// TwinCAT 3 PLC project PLC1
// Title: TcHAL
// Company: none
// Author: Tobias Freyermuth
// ProjectVersion: 0.1.4
// Description: Hardware Abstraction Layer of TwinCAT fieldbus devices
// ProgramVersion: 3.1.4024.12
// libraries:
//   Tc2_EtherCAT, * (Beckhoff Automation GmbH)
//   Tc2_Standard, * (Beckhoff Automation GmbH)
//   Tc2_System, * (Beckhoff Automation GmbH)
//   Tc2_Utilities, * (Beckhoff Automation GmbH)
//   Tc3_Module, * (Beckhoff Automation GmbH)
//   TcUnit, * (www.tcunit.org)
// project tree:
//   analog_input/temperature/ EL3202_0010.TcPOU
//   analog_input/voltage/ EL3164.TcPOU
//   analog_input/_internal/ AI_Channel.TcPOU, AI_Voltage_Channel.TcPOU, AI_Temperature_Channel.TcPOU, I_AI_percentage.TcIO (not stored), I_AI_Temperature.TcIO (not stored), I_AI_Voltage.TcIO (not stored)
//   analog_output/voltage/ EL4002.TcPOU (not stored), EL4102.TcPOU (not stored), EL4004.TcPOU (not stored), EL4134.TcPOU (not stored)
//   analog_output/_internal/ AO_Voltage_Channel.TcPOU (not stored), I_AO_Voltage.TcIO (not stored)
//   coupler/ EK1101.TcPOU (not stored)
//   digital_input/ EL1008.TcPOU (not stored), EL1104.TcPOU (not stored), EL1144.TcPOU (not stored), EL1808.TcPOU (not stored), EL1124.TcPOU (not stored), EL1809.TcPOU (not stored)
//   digital_input/_internal/ HAL_DI_Channel.TcPOU (not stored), I_HAL_DI.TcIO (not stored)
//   digital_output/ EL2008.TcPOU (not stored), EL2124.TcPOU (not stored), EL2024_0010.TcPOU (not stored), EL2502.TcPOU (not stored) (excluded from build), EL2595.TcPOU (not stored), EL2612.TcPOU (not stored), EL2521.TcPOU (not stored) (excluded from build), EL2004.TcPOU (not stored), EL2634.TcPOU (not stored), EL2808.TcPOU (not stored), EL2624.TcPOU (not stored), EL2794.TcPOU (not stored)
//   digital_output/_internal/ HAL_DO_Channel.TcPOU (not stored), I_HAL_DO.TcIO (not stored)
//   / HAL_ErrorEnum.TcDUT (not stored), MAIN.TcPOU (not stored), PlcTask.TcTTO (not stored), Settings.TcGVL (not stored), _internal.TcGVL (not stored)
//   InterfaceManager/ InterfaceManager.TcPOU (not stored), InterfaceManager_test.TcPOU (not stored), I_AI_Percentage_register.TcDUT (not stored), I_AO_Voltage_register.TcDUT (not stored), I_AI_Voltage_register.TcDUT (not stored), I_InterfaceManager.TcIO (not stored)
//   Project Information/ F_GetCompany.TcPOU (not stored), F_GetTitle.TcPOU (not stored), F_GetVersion.TcPOU (not stored)
//   Version/ Global_Version.TcGVL (not stored)
//   _internal/CoE/BeckhoffTerminalConfigEnums/ ENU_DT0800EN02.TcDUT (not stored), ENU_DT0801EN03.TcDUT (not stored)
//   _internal/CoE/buffer/ ring_buffer_CoE_read.TcPOU (not stored)
//   _internal/CoE/ CoE_communication_handler.TcPOU, CoE_property_handler.TcPOU (not stored), CoE_UML_Class Diagram.TcCD (not stored), I_CoE_config_common.TcIO (not stored), I_CoE_property.TcIO, I_CoE_communication_handler.TcIO (not stored)
//   _internal/CoE/properties/ CoE_property.TcPOU
//   _internal/ I_device_control.TcIO (not stored), I_terminal_execution.TcIO (not stored), I_coupler_execution.TcIO (not stored), linear_adc_to_phy.TcPOU (not stored), linear_phy_to_adc.TcPOU (not stored), linear_phy_to_adc_test.TcPOU (not stored), linear_adc_to_phy_test.TcPOU (not stored)

// ---- _internal/CoE/I_CoE_property.TcIO
INTERFACE I_CoE_property

PROPERTY CoE_communication_handler : I_CoE_communication_handler
GET
END_GET
SET
END_SET
END_PROPERTY

PROPERTY dataTypeSize : UDINT
GET
END_GET
END_PROPERTY

METHOD get_value : BOOL
VAR_OUTPUT
    value : Tc2_Utilities.T_Arg ;
	errId : UDINT;
END_VAR
END_METHOD

METHOD handle_read_callback : BOOL
VAR_INPUT
	pt_buffer : POINTER TO Tc2_Utilities.T_Arg;
	errId : UDINT;
END_VAR
END_METHOD

METHOD handle_write_callback : BOOL
VAR_INPUT
	errId : UDINT;
END_VAR
END_METHOD

PROPERTY Index : word
GET
END_GET
END_PROPERTY

PROPERTY init_done : bool
GET
END_GET
END_PROPERTY

PROPERTY PropertyType : E_ArgType
GET
END_GET
SET
END_SET
END_PROPERTY

(**
This method is initializing or reinitializing the property and returns TRUE when this is done.
In case of an error during the init it returns the ErrorCode related to the error that occurred.
*)
METHOD reinit : BOOL
VAR_OUTPUT
	errId: UDINT;
END_VAR
END_METHOD

METHOD run : BOOL
VAR_INPUT
END_VAR
END_METHOD

METHOD set_value : BOOL
VAR_INPUT
    value : Tc2_Utilities.T_Arg ;
END_VAR
END_METHOD

PROPERTY SlaveAddress : UINT
GET
END_GET
SET
END_SET
END_PROPERTY

PROPERTY SubIndex : BYTE
GET
END_GET
END_PROPERTY

PROPERTY valueToWrite : Tc2_Utilities.T_Arg
GET
END_GET
END_PROPERTY

END_INTERFACE

// ---- analog_input/temperature/EL3202_0010.TcPOU
FUNCTION_BLOCK EL3202_0010 IMPLEMENTS I_terminal_execution
VAR_INPUT
END_VAR
VAR_OUTPUT
	AI_Temperature_channel_1 		: I_AI_Temperature :=_channel_1;
	AI_Temperature_channel_2 		: I_AI_Temperature :=_channel_2;
	AI_percent_channe_1				: I_AI_percentage := _channel_1;
	AI_percent_channe_2				: I_AI_percentage := _channel_2;
END_VAR
VAR
// == IO Mapping ==============================================================
	WcState_WcState			AT%I*: BOOL;
	InfoData_State			AT%I*: UINT;
	InfoData_AdsAddr_netId  AT%I*: AMSNETID;
	InfoData_AdsAddr_port 	AT%I*: WORD;
	
	// Channel 1
	RTD_Inputs_Channel_1_Value        			AT%I*: INT;	
	RTD_Inputs_Channel_1_Status_Underrange   	AT%I*: BOOL;
	RTD_Inputs_Channel_1_Status_Overrange   	AT%I*: BOOL;
	RTD_Inputs_Channel_1_Status_Limit_1   		AT%I*: BYTE;
	RTD_Inputs_Channel_1_Status_Limit_2   		AT%I*: BYTE;
	RTD_Inputs_Channel_1_Status_Error   		AT%I*: BOOL;
	RTD_Inputs_Channel_1_Status_TxPDO_State   	AT%I*: BOOL;
	RTD_Inputs_Channel_1_Status_TxPDO_Toggle   	AT%I*: BOOL;
	
	// Channel 2
	RTD_Inputs_Channel_2_Value        			AT%I*: INT;	
	RTD_Inputs_Channel_2_Status_Underrange   	AT%I*: BOOL;
	RTD_Inputs_Channel_2_Status_Overrange   	AT%I*: BOOL;
	RTD_Inputs_Channel_2_Status_Limit_1   		AT%I*: BYTE;
	RTD_Inputs_Channel_2_Status_Limit_2   		AT%I*: BYTE;
	RTD_Inputs_Channel_2_Status_Error   		AT%I*: BOOL;
	RTD_Inputs_Channel_2_Status_TxPDO_State   	AT%I*: BOOL;
	RTD_Inputs_Channel_2_Status_TxPDO_Toggle   	AT%I*: BOOL;
// ============================================================================

	_channel_1 : AI_Temperature_Channel(adc_min:=ADC_MIN, adc_max:=ADC_MAX, physical_min:=PHYSICAL_MIN, physical_max:=PHYSICAL_MAX, channel_number:=1);
	_channel_2 : AI_Temperature_Channel(adc_min:=ADC_MIN, adc_max:=ADC_MAX, physical_min:=PHYSICAL_MIN, physical_max:=PHYSICAL_MAX, channel_number:=2);

    
	// ===============================================================================
	// CoE handling  
	// ==============
    _I_CoE_com_handler      : I_CoE_communication_handler;
    _CoE_prop_handler       : CoE_property_handler;
    // ====  CoE properties  ===========
	_p_DeviceName 			: CoE_property(Index:=16#1008 , SubIndex:=0,PropertyType:=Tc2_Utilities.ARGTYPE_STRING, writable:=FALSE, propertyPullMode:=0, pollingInterval:=T#5S);
	_p_DeviceType 			: CoE_property(Index:=16#1000 , SubIndex:=0,PropertyType:=Tc2_Utilities.ARGTYPE_UDINT, writable:=FALSE, propertyPullMode:=0, pollingInterval:=T#5S);
	_p_ProductCode 			: CoE_property(Index:=16#1018 , SubIndex:=2,PropertyType:=Tc2_Utilities.ARGTYPE_UDINT, writable:=FALSE, propertyPullMode:=0, pollingInterval:=T#5S);
	_p_Revision 			: CoE_property(Index:=16#1018 , SubIndex:=3,PropertyType:=Tc2_Utilities.ARGTYPE_UDINT, writable:=FALSE, propertyPullMode:=0, pollingInterval:=T#5S);
	_p_SerialNumber 		: CoE_property(Index:=16#1018 , SubIndex:=4,PropertyType:=Tc2_Utilities.ARGTYPE_UDINT, writable:=FALSE, propertyPullMode:=0, pollingInterval:=T#5S);
	_p_SoftwareVersion		: CoE_property(Index:=16#100A , SubIndex:=0,PropertyType:=Tc2_Utilities.ARGTYPE_STRING, writable:=FALSE, propertyPullMode:=0, pollingInterval:=T#5S);
	_p_VendorId 			: CoE_property(Index:=16#1018 , SubIndex:=1,PropertyType:=Tc2_Utilities.ARGTYPE_UDINT, writable:=FALSE, propertyPullMode:=0, pollingInterval:=T#5S);
	_p_HardwareVersion		: CoE_property(Index:=16#1009 , SubIndex:=0,PropertyType:=Tc2_Utilities.ARGTYPE_STRING, writable:=FALSE, propertyPullMode:=0, pollingInterval:=T#5S);
	// ==============
	_properties  : ARRAY[1..8]OF I_CoE_property:=[
		_p_DeviceName, _p_DeviceType, _p_ProductCode, _p_Revision, _p_SerialNumber, 
		_p_SoftwareVersion, _p_VendorId, _p_HardwareVersion
	];
	// ===============================================================================
    
    
	_I_InterfaceManager : I_InterfaceManager;
	_terminal_name      : STRING;
	reg_errId           : HAL_ErrorEnum;
	_InitState          : INT;
    neg_wcState: f_trig;
END_VAR
VAR CONSTANT
	ADC_MIN        	: INT:=0;
	ADC_MAX        	: INT:=32767;
	PHYSICAL_MIN 	: INT:=0;
	PHYSICAL_MAX 	: INT:=10;
	
    HARDWARE_REVSION : UINT:=19;
END_VAR

CASE _InitState OF 
	0:  // init parent
        IF _I_InterfaceManager <> 0 AND 
            _I_CoE_com_handler <> 0
        THEN
            _InitState := 5;
		END_IF
		
	5: 
		IF NOT _I_InterfaceManager.register_terminal(terminal_name:=_terminal_name , errId=>reg_errId ) THEN
			RETURN;
		ELSE
			_InitState := 10;
		END_IF
        
	10: // register channel 1 percentage interface 
		IF _I_InterfaceManager.register_I_AI_Percentage(_channel_1, _terminal_name, channel_number := 1, errId=>reg_errId) THEN 
			_InitState := 20;
		END_IF
	20: // register channel 2 percentage interface 
		IF _I_InterfaceManager.register_I_AI_Percentage(_channel_2, _terminal_name, channel_number := 2, errId=>reg_errId) THEN 
			_InitState := 30;
		END_IF

	30: // register channel 1 voltage interface 
		IF _I_InterfaceManager.register_I_AI_Percentage(_channel_1, _terminal_name, channel_number := 1, errId=>reg_errId) THEN 
			_InitState := 40;
		END_IF
		
	40: // register channel 2 voltage interface 
		IF _I_InterfaceManager.register_I_AI_Percentage(_channel_2, _terminal_name, channel_number := 2, errId=>reg_errId) THEN 
			_InitState := 50;
		END_IF
ELSE
	// Channel 1
	_channel_1.wcState							:= WcState_WcState;
	_channel_1.terminal_value 					:= RTD_Inputs_Channel_1_Value;
	_channel_1.io_status_Underrange 			:= RTD_Inputs_Channel_1_Status_Underrange;
	_channel_1.io_status_Overrange 				:= RTD_Inputs_Channel_1_Status_Overrange;
	_channel_1.io_status_Limit_1_greater_value 	:= RTD_Inputs_Channel_1_Status_Limit_1.0;
	_channel_1.io_status_Limit_1_smaller_value	:= RTD_Inputs_Channel_1_Status_Limit_1.1;
	_channel_1.io_status_Limit_2_greater_value 	:= RTD_Inputs_Channel_1_Status_Limit_2.0;
	_channel_1.io_status_Limit_2_smaller_value	:= RTD_Inputs_Channel_1_Status_Limit_2.1;
	_channel_1.io_status_Error 					:= RTD_Inputs_Channel_1_Status_Error;
	_channel_1.io_status_TxPDO_State 			:= RTD_Inputs_Channel_1_Status_TxPDO_State;
	_channel_1.io_status_TxPDO_Toggle 			:= RTD_Inputs_Channel_1_Status_TxPDO_Toggle;
	
	// Channel 2
	_channel_2.wcState							:= WcState_WcState;
	_channel_2.terminal_value 					:= RTD_Inputs_Channel_2_Value;
	_channel_2.io_status_Underrange 			:= RTD_Inputs_Channel_2_Status_Underrange;
	_channel_2.io_status_Overrange 				:= RTD_Inputs_Channel_2_Status_Overrange;
	_channel_2.io_status_Limit_1_greater_value 	:= RTD_Inputs_Channel_2_Status_Limit_1.0;
	_channel_2.io_status_Limit_1_smaller_value	:= RTD_Inputs_Channel_2_Status_Limit_1.1;
	_channel_2.io_status_Limit_2_greater_value 	:= RTD_Inputs_Channel_2_Status_Limit_2.0;
	_channel_2.io_status_Limit_2_smaller_value	:= RTD_Inputs_Channel_2_Status_Limit_2.1;
	_channel_2.io_status_Error 					:= RTD_Inputs_Channel_2_Status_Error;
	_channel_2.io_status_TxPDO_State 			:= RTD_Inputs_Channel_2_Status_TxPDO_State;
	_channel_2.io_status_TxPDO_Toggle 			:= RTD_Inputs_Channel_2_Status_TxPDO_Toggle;

	_channel_1(terminal_address:=InfoData_AdsAddr_port, CoE_communication_handler:=_I_CoE_com_handler);
	_channel_2(terminal_address:=InfoData_AdsAddr_port, CoE_communication_handler:=_I_CoE_com_handler);
END_CASE

_CoE_prop_handler(terminal_address:=InfoData_AdsAddr_port, CoE_communication_handler:=_I_CoE_com_handler, CoE_properties:=_properties);

neg_wcState(CLK:=WcState_WcState);
IF neg_wcState.Q THEN
    ;
END_IF

METHOD FB_init : BOOL
VAR_INPUT
	bInitRetains : BOOL; // if TRUE, the retain variables are initialized (warm start / cold start)
	bInCopyCode : BOOL;  // if TRUE, the instance afterwards gets moved into the copy code (online change)
	CoE_communication_handler: I_CoE_communication_handler;
END_VAR
THIS^._I_CoE_com_handler                := CoE_communication_handler;
_channel_1.CoE_communication_handler	:= CoE_communication_handler;
_channel_2.CoE_communication_handler	:= CoE_communication_handler;
END_METHOD

METHOD run : BOOL
THIS^();
END_METHOD

END_FUNCTION_BLOCK

// ---- analog_input/_internal/AI_Temperature_Channel.TcPOU
FUNCTION_BLOCK AI_Temperature_Channel EXTENDS AI_Channel IMPLEMENTS I_AI_Temperature, I_AI_percentage
VAR
	//  ====  I_AI_percentage  ====
	_max_value 	: REAL:=10.0;
	_min_value 	: REAL:=0.0;
	_value: REAL;
	
	_errId: HAL_ErrorEnum;
    _rValue			: REAL;
    neg_wcState: f_trig;
END_VAR

PROPERTY errId : HAL_ErrorEnum
GET
errId := _errId;
END_GET
END_PROPERTY

PROPERTY max_value : REAL
GET
max_value := _max_value;
END_GET
SET
IF max_value <= 0 THEN
	_max_value := 0.0001;
ELSE
	_max_value := max_value;
END_IF
END_SET
END_PROPERTY

PROPERTY min_value : REAL
GET
min_value := _min_value;
END_GET
SET
_min_value := min_value;
END_SET
END_PROPERTY

PROPERTY rValue : REAL
GET
rValue:=_rValue;
END_GET
SET
IF rValue < DINT_TO_REAL(_physical_min) THEN
	_errId := 6;
ELSIF rValue > DINT_TO_REAL(_physical_max) THEN
	_errId := 7;
ELSE
	_rValue := rValue;
END_IF
END_SET
END_PROPERTY

PROPERTY terminal_value : int
SET
linear_adc_to_phy(
	physical_min	:= _physical_min, 
	physical_max	:= _physical_max, 
	adc_min			:= _adc_min, 
	adc_max			:= _adc_max, 
	adc_value		:= terminal_value, 
	physical_value	=> _rValue, 
	errId			=> _errId
);

linear_adc_to_phy(
	physical_min	:= 0, 
	physical_max	:= 100, 
	adc_min			:= REAL_TO_DINT(_min_value), 
	adc_max			:= REAL_TO_DINT(_max_value), 
	adc_value		:= REAL_TO_DINT(_rValue), 
	physical_value	=> _value, 
	errId			=> _errId
);
END_SET
END_PROPERTY

PROPERTY value : REAL
GET
value := _value;
END_GET
END_PROPERTY

END_FUNCTION_BLOCK

// ---- analog_input/_internal/AI_Channel.TcPOU
FUNCTION_BLOCK AI_Channel
VAR_INPUT
	terminal_address		: WORD;
	CoE_communication_handler	: I_CoE_communication_handler;
END_VAR
VAR_OUTPUT
END_VAR
VAR
	_adc_min        : INT;
    _adc_max        : INT;
	_physical_min 	: INT;
	_physical_max 	: INT;
	_channel_number : UINT;
	_wcState		: BOOL;
	
	// ===============================================================================
	// CoE handling  
    // ==============
    _CoE_prop_handler      : CoE_property_handler;
    _CoE_channel_offset     : INT;
    index_1 				: WORD:= 16#8000 + INT_TO_WORD(_CoE_channel_offset);	
    // ====  CoE properties  ===========
	_p_Enable_user_scale    		: CoE_property(Index:=index_1 , SubIndex:=1, PropertyType:=Tc2_Utilities.ARGTYPE_BOOL, writable:=TRUE, propertyPullMode:=0, pollingInterval:=T#5S);
	_p_Presentation 				: CoE_property(Index:=index_1 , SubIndex:=2, PropertyType:=Tc2_Utilities.ARGTYPE_USINT, writable:=TRUE, propertyPullMode:=0, pollingInterval:=T#5S);			// DT0800EN03
	_p_Watchdog 					: CoE_property(Index:=index_1 , SubIndex:=5, PropertyType:=Tc2_Utilities.ARGTYPE_USINT, writable:=TRUE, propertyPullMode:=0, pollingInterval:=T#5S);			// DT0801EN02
	_p_Enable_user_calibration  	: CoE_property(Index:=index_1 , SubIndex:=7, PropertyType:=Tc2_Utilities.ARGTYPE_BOOL, writable:=TRUE, propertyPullMode:=0, pollingInterval:=T#5S);
	_p_Enable_vendor_calibration    : CoE_property(Index:=index_1 , SubIndex:=8, PropertyType:=Tc2_Utilities.ARGTYPE_BOOL, writable:=TRUE, propertyPullMode:=0, pollingInterval:=T#5S);
	_p_Offset   					: CoE_property(Index:=index_1 , SubIndex:=17, PropertyType:=Tc2_Utilities.ARGTYPE_INT, writable:=TRUE, propertyPullMode:=0, pollingInterval:=T#5S);
	_p_Gain 						: CoE_property(Index:=index_1 , SubIndex:=18, PropertyType:=Tc2_Utilities.ARGTYPE_DINT, writable:=TRUE, propertyPullMode:=0, pollingInterval:=T#5S);
	_p_Default_output   			: CoE_property(Index:=index_1 , SubIndex:=19, PropertyType:=Tc2_Utilities.ARGTYPE_INT, writable:=TRUE, propertyPullMode:=0, pollingInterval:=T#5S);
	_p_Default_output_ramp  		: CoE_property(Index:=index_1 , SubIndex:=20, PropertyType:=Tc2_Utilities.ARGTYPE_UINT, writable:=TRUE, propertyPullMode:=0, pollingInterval:=T#5S);
	_p_User_calibration_offset  	: CoE_property(Index:=index_1 , SubIndex:=21, PropertyType:=Tc2_Utilities.ARGTYPE_INT, writable:=TRUE, propertyPullMode:=0, pollingInterval:=T#5S);
	_p_User_calibration_gain    	: CoE_property(Index:=index_1 , SubIndex:=22, PropertyType:=Tc2_Utilities.ARGTYPE_UINT, writable:=TRUE, propertyPullMode:=0, pollingInterval:=T#5S);
	// ==============
	_properties  : ARRAY[1..11]OF I_CoE_property:=[
		_p_Enable_user_scale, _p_Presentation, _p_Watchdog, _p_Enable_user_calibration, _p_Enable_vendor_calibration, _p_Offset,
		_p_Gain, _p_Default_output, _p_Default_output_ramp, _p_User_calibration_offset, _p_User_calibration_gain];
	// ===============================================================================
    neg_wcState: f_trig;
END_VAR

// CoE Property handling 
_CoE_prop_handler(terminal_address:=terminal_address, CoE_communication_handler:=CoE_communication_handler, CoE_properties:=_properties);

neg_wcState(CLK:=_wcState);
IF neg_wcState.Q THEN
    ;
END_IF

METHOD FB_init : BOOL
VAR_INPUT
	bInitRetains 	: BOOL; // if TRUE, the retain variables are initialized (warm start / cold start)
	bInCopyCode 	: BOOL;  // if TRUE, the instance afterwards gets moved into the copy code (online change)
    adc_min         : INT;
    adc_max         : INT;
	physical_min 	: INT;
	physical_max 	: INT;
	channel_number  : UINT;
END_VAR

VAR
	i: UINT;
END_VAR

_adc_min        := adc_min;
_adc_max        := adc_max;
_physical_min 	:= physical_min;
_physical_max 	:= physical_max;
_channel_number :=channel_number;

CASE channel_number OF
	1:
		_CoE_channel_offset:=16#0;
	2:
		_CoE_channel_offset:=16#10;
	3:
		_CoE_channel_offset:=16#20;
	4:
		_CoE_channel_offset:=16#30;
END_CASE
END_METHOD

METHOD get_Default_output : BOOL
VAR
    targ_value : Tc2_Utilities.T_Arg;
END_VAR
VAR_OUTPUT
	value	: INT;
END_VAR
get_Default_output:=_p_Default_output.get_value(value=>targ_value, errId => );
IF get_Default_output THEN
    MEMCPY(ADR(value), targ_value.pData, targ_value.cbLen);
END_IF
END_METHOD

METHOD get_Default_output_ramp : BOOL
VAR
    targ_value : Tc2_Utilities.T_Arg;
END_VAR
VAR_OUTPUT
	value	: UINT;
END_VAR
get_Default_output_ramp:=_p_Default_output_ramp.get_value(value=>targ_value, errId => );
IF get_Default_output_ramp THEN
    MEMCPY(ADR(value), targ_value.pData, targ_value.cbLen);
END_IF
END_METHOD

METHOD get_Enable_user_calibration : BOOL
VAR
    targ_value : Tc2_Utilities.T_Arg;
END_VAR
VAR_OUTPUT
	value	: BOOL;
END_VAR
get_Enable_user_calibration:=_p_Enable_user_calibration.get_value(value=>targ_value, errId => );
IF get_Enable_user_calibration THEN
    MEMCPY(ADR(value), targ_value.pData, targ_value.cbLen);
END_IF
END_METHOD

METHOD get_Enable_user_scale : BOOL
VAR
    targ_value : Tc2_Utilities.T_Arg;
END_VAR
VAR_OUTPUT
	value	: BOOL;
END_VAR
get_Enable_user_scale:=_p_Enable_user_scale.get_value(value=>targ_value, errId => );
IF get_Enable_user_scale THEN
    MEMCPY(ADR(value), targ_value.pData, targ_value.cbLen);
END_IF
END_METHOD

METHOD get_Enable_vendor_calibration : BOOL
VAR
    targ_value : Tc2_Utilities.T_Arg;
END_VAR
VAR_OUTPUT
	value	: BOOL;
END_VAR
get_Enable_vendor_calibration:=_p_Enable_vendor_calibration.get_value(value=>targ_value, errId => );
IF get_Enable_vendor_calibration THEN
    MEMCPY(ADR(value), targ_value.pData, targ_value.cbLen);
END_IF
END_METHOD

METHOD get_Gain : BOOL
VAR
    targ_value : Tc2_Utilities.T_Arg;
END_VAR
VAR_OUTPUT
	value	: DINT;
END_VAR
get_Gain:=_p_Gain.get_value(value=>targ_value, errId => );
IF get_Gain THEN
    MEMCPY(ADR(value), targ_value.pData, targ_value.cbLen);
END_IF
END_METHOD

METHOD get_Offset : BOOL
VAR
    targ_value : Tc2_Utilities.T_Arg;
END_VAR
VAR_OUTPUT
	value	: INT;
END_VAR
get_Offset:=_p_Offset.get_value(value=>targ_value, errId => );
IF get_Offset THEN
    MEMCPY(ADR(value), targ_value.pData, targ_value.cbLen);
END_IF
END_METHOD

METHOD get_Presentation : BOOL
VAR
	usint_value: USINT;
    targ_value : Tc2_Utilities.T_Arg;
END_VAR
VAR_OUTPUT
	value	: ENU_DT0801EN03;
END_VAR
get_Presentation:=_p_Presentation.get_value(value=>targ_value, errId => );
IF get_Presentation THEN
    MEMCPY(ADR(usint_value), targ_value.pData, targ_value.cbLen);
    value:=USINT_TO_INT(usint_value);
END_IF
END_METHOD

METHOD get_User_calibration_gain : BOOL
VAR
    targ_value : Tc2_Utilities.T_Arg;
END_VAR
VAR_OUTPUT
	value	: UINT;
END_VAR
get_User_calibration_gain:=_p_User_calibration_gain.get_value(value=>targ_value, errId => );
IF get_User_calibration_gain THEN
    MEMCPY(ADR(value), targ_value.pData, targ_value.cbLen);
END_IF
END_METHOD

METHOD get_User_calibration_offset : BOOL
VAR
    targ_value : Tc2_Utilities.T_Arg;
END_VAR
VAR_OUTPUT
	value	: INT;
END_VAR
get_User_calibration_offset:=_p_User_calibration_offset.get_value(value=>targ_value, errId => );
IF get_User_calibration_offset THEN
    MEMCPY(ADR(value), targ_value.pData, targ_value.cbLen);
END_IF
END_METHOD

METHOD get_Watchdog : BOOL
VAR
	usint_value: USINT;
    targ_value : Tc2_Utilities.T_Arg;
END_VAR
VAR_OUTPUT
	value	: ENU_DT0800EN02;
END_VAR
get_Watchdog:=_p_Watchdog.get_value(value=>targ_value, errId => );
IF get_Watchdog THEN
    MEMCPY(ADR(usint_value), targ_value.pData, targ_value.cbLen);
    value:=USINT_TO_INT(usint_value);
END_IF
END_METHOD

PROPERTY io_status_Error : bool
GET
END_GET
SET
END_SET
END_PROPERTY

PROPERTY io_status_Limit_1_greater_value : bool
GET
END_GET
SET
END_SET
END_PROPERTY

PROPERTY io_status_Limit_1_smaller_value : bool
GET
END_GET
SET
END_SET
END_PROPERTY

PROPERTY io_status_Limit_2_greater_value : bool
GET
END_GET
SET
END_SET
END_PROPERTY

PROPERTY io_status_Limit_2_smaller_value : bool
GET
END_GET
SET
END_SET
END_PROPERTY

PROPERTY io_status_Overrange : bool
GET
END_GET
SET
END_SET
END_PROPERTY

PROPERTY io_status_Sync_error : bool
GET
END_GET
SET
END_SET
END_PROPERTY

PROPERTY io_status_TxPDO_State : bool
GET
END_GET
SET
END_SET
END_PROPERTY

PROPERTY io_status_TxPDO_Toggle : bool
GET
END_GET
SET
END_SET
END_PROPERTY

PROPERTY io_status_Underrange : bool
GET
END_GET
SET
END_SET
END_PROPERTY

METHOD set_Default_output : BOOL
VAR_INPUT
	value	: INT;
END_VAR
set_Default_output:=_p_Default_output.set_value(value:=Tc2_Utilities.F_INT(in:=value));
END_METHOD

METHOD set_Default_output_ramp : BOOL
VAR_INPUT
	value	: UINT;
END_VAR
set_Default_output_ramp:=_p_Default_output_ramp.set_value(value:=Tc2_Utilities.F_UINT(in:=value));
END_METHOD

METHOD set_Enable_user_calibration : BOOL
VAR_INPUT
	value	: BOOL;
END_VAR
set_Enable_user_calibration:=_p_Enable_user_calibration.set_value(value:=Tc2_Utilities.F_BOOL(in:=value));
END_METHOD

METHOD set_Enable_user_scale : BOOL
VAR_INPUT
	value	: BOOL;
END_VAR
set_Enable_user_scale:=_p_Enable_user_scale.set_value(value:=Tc2_Utilities.F_BOOL(in:=value));
END_METHOD

METHOD set_Enable_vendor_calibration : BOOL
VAR_INPUT
	value	: BOOL;
END_VAR
set_Enable_vendor_calibration:=_p_Enable_vendor_calibration.set_value(value:=Tc2_Utilities.F_BOOL(in:=value));
END_METHOD

METHOD set_Gain : BOOL
VAR_INPUT
	value	: DINT;
END_VAR
set_Gain:=_p_Gain.set_value(value:=Tc2_Utilities.F_DINT(in:=value));
END_METHOD

METHOD set_Offset : BOOL
VAR_INPUT
	value	: INT;
END_VAR
set_Offset:=_p_Offset.set_value(value:=Tc2_Utilities.F_INT(in:=value));
END_METHOD

METHOD set_Presentation : BOOL
VAR_INPUT
	value	: ENU_DT0801EN03;
END_VAR
VAR
    usint_value : USINT;
END_VAR
usint_value := INT_TO_USINT(value);
set_Presentation:=_p_Presentation.set_value(value:=Tc2_Utilities.F_USINT(in:=usint_value));
END_METHOD

METHOD set_User_calibration_gain : BOOL
VAR_INPUT
	value	: UINT;
END_VAR
set_User_calibration_gain:=_p_User_calibration_gain.set_value(value:=Tc2_Utilities.F_UINT(in:=value));
END_METHOD

METHOD set_User_calibration_offset : BOOL
VAR_INPUT
	value	: INT;
END_VAR
set_User_calibration_offset:=_p_User_calibration_offset.set_value(value:=Tc2_Utilities.F_INT(in:=value));
END_METHOD

METHOD set_Watchdog : BOOL
VAR_INPUT
	value	: ENU_DT0800EN02;
END_VAR
VAR
    usint_value : USINT;
END_VAR
usint_value := INT_TO_USINT(value);
set_Watchdog:=_p_Watchdog.set_value(value:=Tc2_Utilities.F_USINT(in:=usint_value));
END_METHOD

PROPERTY wcState : bool
GET
wcState:=_wcState;
END_GET
SET
_wcState:=wcState;
END_SET
END_PROPERTY

END_FUNCTION_BLOCK

// ---- _internal/CoE/CoE_communication_handler.TcPOU
(**
This function bock handles ADS read and write requests.
To read or write an ADS property pass an object that implements the "I_CoE_property" interface through the "add_read_request" or "add_write_request" method.
All requests will be added to an internal read or write buffer and executed one by one.
The object will be updated through the callback interface when the read or write process is done.
*)
FUNCTION_BLOCK CoE_communication_handler IMPLEMENTS I_CoE_communication_handler
VAR_INPUT
	amsNetId	: T_AmsNetId;
END_VAR
VAR_OUTPUT
END_VAR
VAR
	// ==  read  ================================== 
	done_reading_coe		: f_trig;
	CoE_property_to_read	: I_CoE_property;
	read_requests_table 	: ring_buffer_CoE_read; 
	
	coe_read 	: FB_EcCoESdoRead;	
	
	_readState		: INT;
	_executeRead	: BOOL;
	_readBuffer		: Tc2_Utilities.T_Arg;
	
	// ==  write  ================================== 
	done_writing_coe		: f_trig;
	CoE_property_to_write	: I_CoE_property;
	write_requests_table 	: ring_buffer_CoE_read; 
	
	coe_write 	: FB_EcCoESdoWrite;	
	
	_writeState			: INT;
	_executeWrite		: BOOL;
	_writeBuffer		: Tc2_Utilities.T_Arg;

END_VAR

// ===========================
// handle read requests
// ===
CASE _readState OF 
	0:
		IF read_requests_table.read(data=> CoE_property_to_read)THEN 
			_executeRead := TRUE;
			_readState := 10;			
		END_IF

	10:
		IF done_reading_coe.q THEN
			CoE_property_to_read.handle_read_callback(pt_buffer:=_readBuffer.pData, errId:=coe_read.nErrId);
			_executeRead:=FALSE;
			_readState := 0;
		END_IF
ELSE
	_readState := 0;
END_CASE

IF CoE_property_to_read <> 0 THEN
    _readBuffer.eType := CoE_property_to_read.PropertyType;
	coe_read(
		sNetId		:= amsNetId, 
		nSlaveAddr	:= CoE_property_to_read.SlaveAddress, 
		nSubIndex	:= CoE_property_to_read.SubIndex, 
		nIndex		:= CoE_property_to_read.Index, 
		pDstBuf		:= _readBuffer.pData, 
		cbBufLen	:= _readBuffer.cbLen, 
		bExecute	:= _executeRead, 
		tTimeout	:= , 
		bBusy		=> , 
		bError		=> , 
		nErrId		=> , 
		cbRead		=> );
		
	done_reading_coe(clk:=coe_read.bBusy);
END_IF


// ===========================
// hadndle write requests
// ===
CASE _writeState OF 
	0:
		IF write_requests_table.read(data=> CoE_property_to_write) THEN 
			_writeBuffer := CoE_property_to_write.valueToWrite;
			_executeWrite := TRUE;
			_writeState := 10;			
		END_IF

	10:
		IF done_writing_coe.q THEN
			CoE_property_to_write.handle_write_callback(errId:=coe_write.nErrId);
			_executeWrite:=FALSE;
			_writeState := 0;
		END_IF
ELSE
	_readState := 0;
END_CASE

IF CoE_property_to_write <> 0 THEN
	coe_write(
		sNetId		:= amsNetId, 
		nSlaveAddr	:= CoE_property_to_write.SlaveAddress, 
		nSubIndex	:= CoE_property_to_write.SubIndex, 
		nIndex		:= CoE_property_to_write.Index, 
		pSrcBuf		:= _writeBuffer.pData, 
		cbBufLen	:= CoE_property_to_write.dataTypeSize, 
		bExecute	:= _executeWrite, 
		tTimeout	:= , 
		bBusy		=> , 
		bError		=> , 
		nErrId		=> );
		
	done_writing_coe(clk:=coe_write.bBusy);
END_IF
// ===========================

METHOD add_read_request : BOOL
VAR_INPUT
	request	: I_CoE_property;
END_VAR

IF request <> 0 THEN
	add_read_request:= THIS^.read_requests_table.write(request);
ELSE
	add_read_request:=FALSE;
END_IF
END_METHOD

METHOD add_write_request : BOOL
VAR_INPUT
	request	: I_CoE_property;
END_VAR

IF request <> 0 THEN
	add_write_request:= THIS^.write_requests_table.write(request);
ELSE
	add_write_request:=FALSE;
END_IF
END_METHOD

END_FUNCTION_BLOCK

// ---- _internal/CoE/properties/CoE_property.TcPOU
FUNCTION_BLOCK CoE_property IMPLEMENTS I_CoE_property
VAR_INPUT
END_VAR
VAR_OUTPUT
END_VAR
VAR
	_SubIndex 		: BYTE;
	_Index			: WORD;
    _propertyType : Tc2_Utilities.E_ArgType := Tc2_Utilities.ARGTYPE_UNKNOWN;
	_init_done		: BOOL;
	_neg_replay		: f_trig;
	_SlaveAddress	: WORD;
	_propertyPullMode	: UINT;
	_pollingInterval: TIME;
	_I_CoE_communication_handler: I_CoE_communication_handler;
	
	_read_errId		: UDINT;
	_write_errId	: UDINT;
	_init_state		: INT;
	
	_valueToWrite 	: Tc2_Utilities.T_Arg;
    _value : Tc2_Utilities.T_Arg;

	pollingTimer: ton;
	
	errId: INT;
END_VAR

CASE _propertyPullMode OF 
	0:  // cashed 
		;
	
	1:  // polling 
		pollingTimer(IN:=NOT pollingTimer.q, PT:=_pollingInterval);
		IF pollingTimer.Q THEN
			IF THIS^._I_CoE_communication_handler <> 0 THEN 
				THIS^._I_CoE_communication_handler.add_read_request(THIS^);
			ELSE
				errId:=1;
			END_IF
		END_IF
	
	2: // on request
		IF THIS^._I_CoE_communication_handler <> 0 THEN 
			THIS^._I_CoE_communication_handler.add_read_request(THIS^);
		ELSE
			errId:=1; 
		END_IF

ELSE
	errId:=2; 
END_CASE

PROPERTY CoE_communication_handler : I_CoE_communication_handler
GET
CoE_communication_handler:=_I_CoE_communication_handler;
END_GET
SET
_I_CoE_communication_handler:=CoE_communication_handler;
END_SET
END_PROPERTY

PROPERTY dataTypeSize : UDINT
GET
dataTypeSize := _value.cbLen;
END_GET
END_PROPERTY

METHOD FB_init : BOOL
VAR_INPUT
	bInitRetains 			: BOOL; // if TRUE, the retain variables are initialized (warm start / cold start)
	bInCopyCode 			: BOOL;  // if TRUE, the instance afterwards gets moved into the copy code (online change)
	Index					: WORD;
	SubIndex				: BYTE;
    propertyType : Tc2_Utilities.E_ArgType;
	writable				: BOOL;
	propertyPullMode			: UINT;
	pollingInterval 		: TIME;
END_VAR
_Index:=Index;
_SubIndex:=SubIndex;
_propertyType:=propertyType;
_propertyPullMode:=propertyPullMode;
_pollingInterval:=pollingInterval;
END_METHOD

METHOD get_value : BOOL
VAR_OUTPUT
	value : Tc2_Utilities.T_Arg ;
	errId : UDINT;
END_VAR
IF init_done THEN
        IF _value.eType=THIS^.PropertyType THEN
        value := _value;
        get_value := TRUE;
    ELSE
        errId := 400;
        get_value := FALSE;
	END_IF
ELSE
	errId := 2;
	get_value := FALSE;
END_IF
END_METHOD

METHOD handle_read_callback : BOOL
VAR_INPUT
	pt_buffer : POINTER TO Tc2_Utilities.T_Arg;
	errId : UDINT;
END_VAR
_value := pt_buffer^;
_init_done:=TRUE;
_read_errId:=errId;
END_METHOD

METHOD handle_write_callback : BOOL
VAR_INPUT
	errId : UDINT;
END_VAR
_write_errId:=errId;
END_METHOD

PROPERTY Index : word
GET
Index:=_Index;
END_GET
SET
_Index:=Index;
END_SET
END_PROPERTY

PROPERTY init_done : BOOL
GET
init_done := _init_done;
END_GET
END_PROPERTY

PROPERTY PropertyType : E_ArgType
GET
PropertyType:=_propertyType;
END_GET
SET
_propertyType:=PropertyType;
END_SET
END_PROPERTY

METHOD reinit : BOOL
VAR_OUTPUT
	errId: UDINT;
END_VAR

CASE _init_state OF 
	0:  // add read request and continue
		_init_done:=FALSE;
		reinit:=FALSE;
		IF THIS^._I_CoE_communication_handler <> 0 THEN 
			THIS^._I_CoE_communication_handler.add_read_request(THIS^);
		ELSE
			errId:=1;
		END_IF
		_init_state := 10;
		
	10: // wait for read callback
		reinit:=TRUE;
		errId:=_read_errId;
		_init_state := 0;
END_CASE
END_METHOD

METHOD run : BOOL
THIS^();
END_METHOD

METHOD set_value : BOOL
VAR_INPUT
	value : Tc2_Utilities.T_Arg ;
END_VAR
IF value.eType=THIS^.PropertyType THEN
    _valueToWrite := value;
    IF THIS^._I_CoE_communication_handler <> 0 THEN 
        THIS^._I_CoE_communication_handler.add_write_request(THIS^);
        set_value := TRUE;
    ELSE
        set_value := FALSE;
        errId:=1;
    END_IF
ELSE
    set_value := FALSE;
    errId := 400;
END_IF
END_METHOD

PROPERTY SlaveAddress : uint
GET
SlaveAddress:=_SlaveAddress;
END_GET
SET
_SlaveAddress:=SlaveAddress;
END_SET
END_PROPERTY

PROPERTY SubIndex : BYTE
GET
SubIndex:=_SubIndex;
END_GET
SET
_SubIndex:=SubIndex;
END_SET
END_PROPERTY

PROPERTY valueToWrite : Tc2_Utilities.T_Arg
GET
valueToWrite := _valueToWrite;
END_GET
END_PROPERTY

END_FUNCTION_BLOCK

// ---- analog_input/voltage/EL3164.TcPOU
(**
This function block abstracts the Beckhoff EtherCAT terminal EL3164 (0…10 V, 16 Bit)
*)
FUNCTION_BLOCK EL3164 IMPLEMENTS I_terminal_execution
VAR_INPUT
END_VAR
VAR_OUTPUT
	AI_Voltage_channel_1 		: I_AI_Voltage :=_channel_1;
	AI_Voltage_channel_2 		: I_AI_Voltage :=_channel_2;
	AI_Voltage_channel_3 		: I_AI_Voltage :=_channel_3;
	AI_Voltage_channel_4 		: I_AI_Voltage :=_channel_4;
	AI_percent_channe_1			: I_AI_percentage := _channel_1;
	AI_percent_channe_2			: I_AI_percentage := _channel_2;
	AI_percent_channe_3			: I_AI_percentage := _channel_3;
	AI_percent_channe_4			: I_AI_percentage := _channel_4;
END_VAR
VAR
// == IO Mapping ==============================================================
// The channel status Limits 1 and 2 have to be defined as BYTE since they are 
// of BIT2 in the terminal, but there is no such datatype in the PLC.

	WcState_WcState			AT%I*: BOOL;
	InfoData_State			AT%I*: UINT;
	InfoData_AdsAddr_netId  AT%I*: AMSNETID;
	InfoData_AdsAddr_port 	AT%I*: WORD;
	
	// Channel 1
	AI_Standard_Channel_1_Value        			AT%I*: INT;	
	AI_Standard_Channel_1_Status_Underrange   	AT%I*: BOOL;
	AI_Standard_Channel_1_Status_Overrange   	AT%I*: BOOL;
	AI_Standard_Channel_1_Status_Limit_1   		AT%I*: BYTE;
	AI_Standard_Channel_1_Status_Limit_2   		AT%I*: BYTE;
	AI_Standard_Channel_1_Status_Error   		AT%I*: BOOL;
	AI_Standard_Channel_1_Status_Sync_error   	AT%I*: BOOL;
	AI_Standard_Channel_1_Status_TxPDO_State   	AT%I*: BOOL;
	AI_Standard_Channel_1_Status_TxPDO_Toggle   AT%I*: BOOL;

	// Channel 2
	AI_Standard_Channel_2_Value        			AT%I*: INT;	
	AI_Standard_Channel_2_Status_Underrange   	AT%I*: BOOL;
	AI_Standard_Channel_2_Status_Overrange   	AT%I*: BOOL;
	AI_Standard_Channel_2_Status_Limit_1   		AT%I*: BYTE;
	AI_Standard_Channel_2_Status_Limit_2   		AT%I*: BYTE;
	AI_Standard_Channel_2_Status_Error   		AT%I*: BOOL;
	AI_Standard_Channel_2_Status_Sync_error   	AT%I*: BOOL;
	AI_Standard_Channel_2_Status_TxPDO_State   	AT%I*: BOOL;
	AI_Standard_Channel_2_Status_TxPDO_Toggle   AT%I*: BOOL;
	
	// Channel 3
	AI_Standard_Channel_3_Value        			AT%I*: INT;	
	AI_Standard_Channel_3_Status_Underrange   	AT%I*: BOOL;
	AI_Standard_Channel_3_Status_Overrange   	AT%I*: BOOL;
	AI_Standard_Channel_3_Status_Limit_1   		AT%I*: BYTE;
	AI_Standard_Channel_3_Status_Limit_2   		AT%I*: BYTE;
	AI_Standard_Channel_3_Status_Error   		AT%I*: BOOL;
	AI_Standard_Channel_3_Status_Sync_error   	AT%I*: BOOL;
	AI_Standard_Channel_3_Status_TxPDO_State   	AT%I*: BOOL;
	AI_Standard_Channel_3_Status_TxPDO_Toggle   AT%I*: BOOL;
	
	// Channel 4
	AI_Standard_Channel_4_Value        			AT%I*: INT;	
	AI_Standard_Channel_4_Status_Underrange   	AT%I*: BOOL;
	AI_Standard_Channel_4_Status_Overrange   	AT%I*: BOOL;
	AI_Standard_Channel_4_Status_Limit_1   		AT%I*: BYTE;  
	AI_Standard_Channel_4_Status_Limit_2   		AT%I*: BYTE;
	AI_Standard_Channel_4_Status_Error   		AT%I*: BOOL;
	AI_Standard_Channel_4_Status_Sync_error   	AT%I*: BOOL;
	AI_Standard_Channel_4_Status_TxPDO_State   	AT%I*: BOOL;
	AI_Standard_Channel_4_Status_TxPDO_Toggle   AT%I*: BOOL;
// ============================================================================

	_channel_1 : AI_Voltage_Channel(adc_min:=ADC_MIN, adc_max:=ADC_MAX, physical_min:=PHYSICAL_MIN, physical_max:=PHYSICAL_MAX, channel_number:=1);
	_channel_2 : AI_Voltage_Channel(adc_min:=ADC_MIN, adc_max:=ADC_MAX, physical_min:=PHYSICAL_MIN, physical_max:=PHYSICAL_MAX, channel_number:=2);
	_channel_3 : AI_Voltage_Channel(adc_min:=ADC_MIN, adc_max:=ADC_MAX, physical_min:=PHYSICAL_MIN, physical_max:=PHYSICAL_MAX, channel_number:=3);
	_channel_4 : AI_Voltage_Channel(adc_min:=ADC_MIN, adc_max:=ADC_MAX, physical_min:=PHYSICAL_MIN, physical_max:=PHYSICAL_MAX, channel_number:=4);
	
    
	// ===============================================================================
	// CoE handling  
	// ==============
    _I_CoE_com_handler      : I_CoE_communication_handler;
    _CoE_prop_handler       : CoE_property_handler;
    // ====  CoE properties  ===========
	_p_DeviceName 			: CoE_property(Index:=16#1008 , SubIndex:=0,PropertyType:=Tc2_Utilities.ARGTYPE_STRING, writable:=FALSE, propertyPullMode:=0, pollingInterval:=T#5S);
	_p_DeviceType 			: CoE_property(Index:=16#1000 , SubIndex:=0,PropertyType:=Tc2_Utilities.ARGTYPE_UDINT, writable:=FALSE, propertyPullMode:=0, pollingInterval:=T#5S);
	_p_ProductCode 			: CoE_property(Index:=16#1018 , SubIndex:=2,PropertyType:=Tc2_Utilities.ARGTYPE_UDINT, writable:=FALSE, propertyPullMode:=0, pollingInterval:=T#5S);
	_p_Revision 			: CoE_property(Index:=16#1018 , SubIndex:=3,PropertyType:=Tc2_Utilities.ARGTYPE_UDINT, writable:=FALSE, propertyPullMode:=0, pollingInterval:=T#5S);
	_p_SerialNumber 		: CoE_property(Index:=16#1018 , SubIndex:=4,PropertyType:=Tc2_Utilities.ARGTYPE_UDINT, writable:=FALSE, propertyPullMode:=0, pollingInterval:=T#5S);
	_p_SoftwareVersion		: CoE_property(Index:=16#100A , SubIndex:=0,PropertyType:=Tc2_Utilities.ARGTYPE_STRING, writable:=FALSE, propertyPullMode:=0, pollingInterval:=T#5S);
	_p_VendorId 			: CoE_property(Index:=16#1018 , SubIndex:=1,PropertyType:=Tc2_Utilities.ARGTYPE_UDINT, writable:=FALSE, propertyPullMode:=0, pollingInterval:=T#5S);
	_p_HardwareVersion		: CoE_property(Index:=16#1009 , SubIndex:=0,PropertyType:=Tc2_Utilities.ARGTYPE_STRING, writable:=FALSE, propertyPullMode:=0, pollingInterval:=T#5S);
	// ==============
	_properties  : ARRAY[1..8]OF I_CoE_property:=[
		_p_DeviceName, _p_DeviceType, _p_ProductCode, _p_Revision, _p_SerialNumber, 
		_p_SoftwareVersion, _p_VendorId, _p_HardwareVersion
	];
	// ===============================================================================
    
    
	_I_InterfaceManager : I_InterfaceManager;
	_terminal_name      : STRING;
	reg_errId           : HAL_ErrorEnum;
	_InitState          : INT;
    neg_wcState: f_trig;
END_VAR
VAR CONSTANT
	ADC_MIN        	: INT:=0;
	ADC_MAX        	: INT:=32767;
	PHYSICAL_MIN 	: INT:=0;
	PHYSICAL_MAX 	: INT:=10;
	
    HARDWARE_REVSION : UINT:=19;
END_VAR


CASE _InitState OF 
	0:  // init parent
        IF _I_InterfaceManager <> 0 AND 
            _I_CoE_com_handler <> 0
        THEN
            _InitState := 5;
		END_IF
		
	5: 
		IF NOT _I_InterfaceManager.register_terminal(terminal_name:=_terminal_name , errId=>reg_errId ) THEN
			RETURN;
		ELSE
			_InitState := 10;
		END_IF
	
	10: // register channel 1 percentage interface 
		IF _I_InterfaceManager.register_I_AI_Percentage(_channel_1, _terminal_name, channel_number := 1, errId=>reg_errId) THEN 
			_InitState := 20;
		END_IF
	20: // register channel 2 percentage interface 
		IF _I_InterfaceManager.register_I_AI_Percentage(_channel_2, _terminal_name, channel_number := 2, errId=>reg_errId) THEN 
			_InitState := 30;
		END_IF
		
	30: // register channel 3 percentage interface 
		IF _I_InterfaceManager.register_I_AI_Percentage(_channel_3, _terminal_name, channel_number := 3, errId=>reg_errId) THEN 
			_InitState := 40;
		END_IF
		
	40: // register channel 4 percentage interface 
		IF _I_InterfaceManager.register_I_AI_Percentage(_channel_4, _terminal_name, channel_number := 4, errId=>reg_errId) THEN 
			_InitState := 50;
		END_IF

	50: // register channel 1 voltage interface 
		IF _I_InterfaceManager.register_I_AI_Voltage(_channel_1, _terminal_name, channel_number := 1, errId=>reg_errId) THEN 
			_InitState := 60;
		END_IF
		
	60: // register channel 2 voltage interface 
		IF _I_InterfaceManager.register_I_AI_Voltage(_channel_2, _terminal_name, channel_number := 2, errId=>reg_errId) THEN 
			_InitState := 70;
		END_IF
		
	70: // register channel 3 voltage interface 
		IF _I_InterfaceManager.register_I_AI_Voltage(_channel_3, _terminal_name, channel_number := 3, errId=>reg_errId) THEN 
			_InitState := 80;
		END_IF
		
	80: // register channel 4 voltage interface 
		IF _I_InterfaceManager.register_I_AI_Voltage(_channel_4, _terminal_name, channel_number := 4, errId=>reg_errId) THEN 
			_InitState := 90;
		END_IF
ELSE
	// Channel 1
	_channel_1.wcState							:= WcState_WcState;	
	_channel_1.terminal_value 					:= AI_Standard_Channel_1_Value;
	_channel_1.io_status_Underrange 			:= AI_Standard_Channel_1_Status_Underrange;
	_channel_1.io_status_Overrange 				:= AI_Standard_Channel_1_Status_Overrange;
	_channel_1.io_status_Limit_1_greater_value 	:= AI_Standard_Channel_1_Status_Limit_1.0;
	_channel_1.io_status_Limit_1_smaller_value	:= AI_Standard_Channel_1_Status_Limit_1.1;
	_channel_1.io_status_Limit_2_greater_value 	:= AI_Standard_Channel_1_Status_Limit_2.0;
	_channel_1.io_status_Limit_2_smaller_value	:= AI_Standard_Channel_1_Status_Limit_2.1;
	_channel_1.io_status_Error 					:= AI_Standard_Channel_1_Status_Error;
	_channel_1.io_status_Sync_error 			:= AI_Standard_Channel_1_Status_Sync_error;
	_channel_1.io_status_TxPDO_State 			:= AI_Standard_Channel_1_Status_TxPDO_State;
	_channel_1.io_status_TxPDO_Toggle 			:= AI_Standard_Channel_1_Status_TxPDO_Toggle;
	
	// Channel 2
	_channel_2.wcState							:= WcState_WcState;
	_channel_2.terminal_value 					:= AI_Standard_Channel_2_Value;
	_channel_2.io_status_Underrange 			:= AI_Standard_Channel_2_Status_Underrange;
	_channel_2.io_status_Overrange 				:= AI_Standard_Channel_2_Status_Overrange;
	_channel_2.io_status_Limit_1_greater_value 	:= AI_Standard_Channel_2_Status_Limit_1.0;
	_channel_2.io_status_Limit_1_smaller_value	:= AI_Standard_Channel_2_Status_Limit_1.1;
	_channel_2.io_status_Limit_2_greater_value 	:= AI_Standard_Channel_2_Status_Limit_2.0;
	_channel_2.io_status_Limit_2_smaller_value	:= AI_Standard_Channel_2_Status_Limit_2.1;
	_channel_2.io_status_Error 					:= AI_Standard_Channel_2_Status_Error;
	_channel_2.io_status_Sync_error 			:= AI_Standard_Channel_2_Status_Sync_error;
	_channel_2.io_status_TxPDO_State 			:= AI_Standard_Channel_2_Status_TxPDO_State;
	_channel_2.io_status_TxPDO_Toggle 			:= AI_Standard_Channel_2_Status_TxPDO_Toggle;

	// Channel 3
	_channel_3.wcState							:= WcState_WcState;
	_channel_3.terminal_value 					:= AI_Standard_Channel_3_Value;
	_channel_3.io_status_Underrange 			:= AI_Standard_Channel_3_Status_Underrange;
	_channel_3.io_status_Overrange 				:= AI_Standard_Channel_3_Status_Overrange;
	_channel_3.io_status_Limit_1_greater_value 	:= AI_Standard_Channel_3_Status_Limit_1.0;
	_channel_3.io_status_Limit_1_smaller_value	:= AI_Standard_Channel_3_Status_Limit_1.1;
	_channel_3.io_status_Limit_2_greater_value 	:= AI_Standard_Channel_3_Status_Limit_2.0;
	_channel_3.io_status_Limit_2_smaller_value	:= AI_Standard_Channel_3_Status_Limit_2.1;
	_channel_3.io_status_Error 					:= AI_Standard_Channel_3_Status_Error;
	_channel_3.io_status_Sync_error 			:= AI_Standard_Channel_3_Status_Sync_error;
	_channel_3.io_status_TxPDO_State 			:= AI_Standard_Channel_3_Status_TxPDO_State;
	_channel_3.io_status_TxPDO_Toggle 			:= AI_Standard_Channel_3_Status_TxPDO_Toggle;

	// Channel 4
	_channel_4.wcState							:= WcState_WcState;	
	_channel_4.terminal_value 					:= AI_Standard_Channel_4_Value;
	_channel_4.io_status_Underrange 			:= AI_Standard_Channel_4_Status_Underrange;
	_channel_4.io_status_Overrange 				:= AI_Standard_Channel_4_Status_Overrange;
	_channel_4.io_status_Limit_1_greater_value 	:= AI_Standard_Channel_4_Status_Limit_1.0;
	_channel_4.io_status_Limit_1_smaller_value	:= AI_Standard_Channel_4_Status_Limit_1.1;
	_channel_4.io_status_Limit_2_greater_value 	:= AI_Standard_Channel_4_Status_Limit_2.0;
	_channel_4.io_status_Limit_2_smaller_value	:= AI_Standard_Channel_4_Status_Limit_2.1;
	_channel_4.io_status_Error 					:= AI_Standard_Channel_4_Status_Error;
	_channel_4.io_status_Sync_error 			:= AI_Standard_Channel_4_Status_Sync_error;
	_channel_4.io_status_TxPDO_State 			:= AI_Standard_Channel_4_Status_TxPDO_State;
	_channel_4.io_status_TxPDO_Toggle 			:= AI_Standard_Channel_4_Status_TxPDO_Toggle;	

	_channel_1(terminal_address:=InfoData_AdsAddr_port, CoE_communication_handler:=_I_CoE_com_handler);
	_channel_2(terminal_address:=InfoData_AdsAddr_port, CoE_communication_handler:=_I_CoE_com_handler);
	_channel_3(terminal_address:=InfoData_AdsAddr_port, CoE_communication_handler:=_I_CoE_com_handler);
	_channel_4(terminal_address:=InfoData_AdsAddr_port, CoE_communication_handler:=_I_CoE_com_handler);
END_CASE


_CoE_prop_handler(terminal_address:=InfoData_AdsAddr_port, CoE_communication_handler:=_I_CoE_com_handler, CoE_properties:=_properties);

neg_wcState(CLK:=WcState_WcState);
IF neg_wcState.Q THEN
    ;
END_IF

METHOD FB_init : BOOL
VAR_INPUT
	bInitRetains : BOOL; // if TRUE, the retain variables are initialized (warm start / cold start)
	bInCopyCode : BOOL;  // if TRUE, the instance afterwards gets moved into the copy code (online change)
	CoE_communication_handler   : I_CoE_communication_handler;
	InterfaceManager            : I_InterfaceManager;
	name                        : STRING;
END_VAR
_I_CoE_com_handler        	            := CoE_communication_handler;
_channel_1.CoE_communication_handler	:= CoE_communication_handler;
_channel_2.CoE_communication_handler	:= CoE_communication_handler;
_channel_3.CoE_communication_handler	:= CoE_communication_handler;
_channel_4.CoE_communication_handler	:= CoE_communication_handler;
_I_InterfaceManager := InterfaceManager;
_terminal_name := name;
END_METHOD

METHOD run : BOOL
THIS^();
END_METHOD

END_FUNCTION_BLOCK

// ---- analog_input/_internal/AI_Voltage_Channel.TcPOU
FUNCTION_BLOCK AI_Voltage_Channel EXTENDS AI_Channel IMPLEMENTS I_AI_Voltage, I_AI_percentage
VAR
	//  ====  I_AI_percentage  ====
	_max_value 	: REAL:=10.0;
	_min_value 	: REAL:=0.0;
	_value: REAL;
	
	_errId: HAL_ErrorEnum;
    _rValue			: REAL;
    neg_wcState: f_trig;
END_VAR

PROPERTY errId : UINT
GET
errId := _errId;
END_GET
END_PROPERTY

PROPERTY max_value : REAL
GET
max_value := _max_value;
END_GET
SET
IF max_value <= 0 THEN
	_max_value := 0.0001;
ELSE
	_max_value := max_value;
END_IF
END_SET
END_PROPERTY

PROPERTY min_value : REAL
GET
min_value := _min_value;
END_GET
SET
_min_value := min_value;
END_SET
END_PROPERTY

PROPERTY rValue : REAL
GET
rValue:=_rValue;
END_GET
SET
IF rValue < DINT_TO_REAL(_physical_min) THEN
	_errId := 6;
ELSIF rValue > DINT_TO_REAL(_physical_max) THEN
	_errId := 7;
ELSE
	_rValue := rValue;
END_IF
END_SET
END_PROPERTY

PROPERTY terminal_value : int
SET
linear_adc_to_phy(
	physical_min	:= _physical_min, 
	physical_max	:= _physical_max, 
	adc_min			:= _adc_min, 
	adc_max			:= _adc_max, 
	adc_value		:= terminal_value, 
	physical_value	=> _rValue, 
	errId			=> _errId
);

linear_adc_to_phy(
	physical_min	:= 0, 
	physical_max	:= 100, 
	adc_min			:= REAL_TO_DINT(_min_value), 
	adc_max			:= REAL_TO_DINT(_max_value), 
	adc_value		:= REAL_TO_DINT(_rValue), 
	physical_value	=> _value, 
	errId			=> _errId
);
END_SET
END_PROPERTY

PROPERTY value : REAL
GET
value := _value;
END_GET
END_PROPERTY

END_FUNCTION_BLOCK
